// TIA Portal V17 export
// export: Created 2025-05-22T06:00:03.08653Z, ExportSetting WithDefaults, DisplayName Totally Integrated Automation Portal, DisplayVersion V17 Update 8, DisplayName TIA Portal Openness, DisplayVersion V17 Update 8, DisplayName TIA Portal Version Control Interface, DisplayVersion V17, DisplayName SINAMICS Startdrive Advanced, DisplayVersion V17 SP2, DisplayName SINAMICS Startdrive G110M, G120, G120C, G120D, G120P, G115D, DisplayVersion V17 SP2, DisplayName SINAMICS Startdrive G130, G150, S120, S150, SINAMICS MV, S210, DisplayVersion V17 SP2, DisplayName STEP 7 Professional, DisplayVersion V17 Update 8, DisplayName SINUMERIK ONE STEP 7 Toolbox, DisplayVersion V17 Update 12, DisplayName SINUMERIK ONE PLC Basic Program Plus, DisplayVersion V17 Update 12, DisplayName SINUMERIK 840D sl STEP 7 Toolbox, DisplayVersion V17 Update 12, DisplayName STEP 7 Safety, DisplayVersion V17 Update 6, DisplayName WinCC Advanced, DisplayVersion V17 Update 8
FUNCTION "FC421_HOLA_PC_ALARM" : Void   // FC421, LAD
{ S7_Optimized_Access := 'FALSE' }
AUTHOR : ETXETAR
VERSION : 1.0
// stored: AutoNumber false, IsIECCheckEnabled false, SetENOAutomatically false, UDAEnableTagReadback false
   VAR_TEMP
      ERROR : Bool;   // ERROR
      ERROR_CODE : Int;   // ERROR CODE
      ZERO : DWord;   // ZERO
      RESET : Struct   // RESET
         DBB_120 : Word;   // RESET $A_DBB[120]
         DBB_122 : Word;   // RESET $A_DBB[122]
         DBB_124 : Word;   // RESET $A_DBB[124]
         DBB_126 : Word;   // RESET $A_DBB[126]
      END_STRUCT;
   END_VAR
   VAR CONSTANT
      READ : Byte := 16#3;
      WRITE : Byte := 16#4;
      FC_NUMBER : DInt := 202;   // FC NUMBER
   END_VAR
   VAR_TEMP   // added for the SCL form of the ladder/FBD networks
      _w1 : Bool;
      _w2 : Bool;
      _w3 : Bool;
   END_VAR
BEGIN

REGION Network 1: CALL FC21 TOOL ALARMS - $A_DBW[120] TO $A_DBW[126] / READ $A_DBB[102-108]
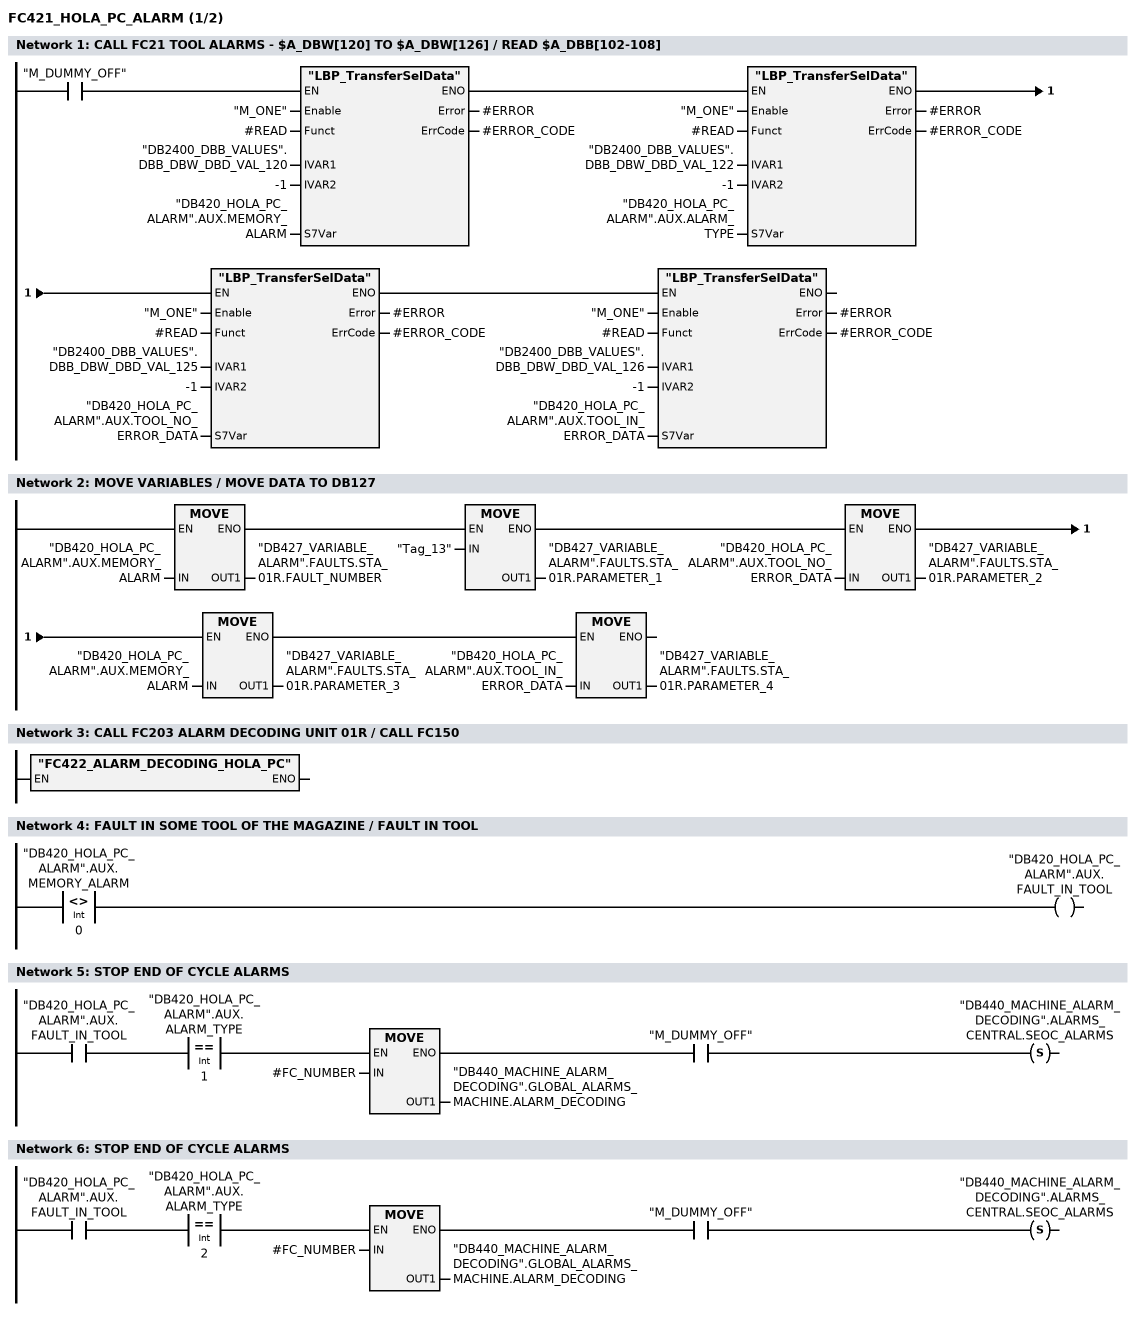
   RUNG wire#powerrail
      Contact( "M_DUMMY_OFF" )
      "LBP_TransferSelData"(Enable := "M_ONE", Funct := #READ, IVAR1 := "DB2400_DBB_VALUES".DBB_DBW_DBD_VAL_120, IVAR2 := -1, S7Var := "DB420_HOLA_PC_ALARM".AUX.MEMORY_ALARM, Error => #ERROR, ErrCode => #ERROR_CODE)
      "LBP_TransferSelData"(Enable := "M_ONE", Funct := #READ, IVAR1 := "DB2400_DBB_VALUES".DBB_DBW_DBD_VAL_122, IVAR2 := -1, S7Var := "DB420_HOLA_PC_ALARM".AUX.ALARM_TYPE, Error => #ERROR, ErrCode => #ERROR_CODE)
      "LBP_TransferSelData"(Enable := "M_ONE", Funct := #READ, IVAR1 := "DB2400_DBB_VALUES".DBB_DBW_DBD_VAL_125, IVAR2 := -1, S7Var := "DB420_HOLA_PC_ALARM".AUX.TOOL_NO_ERROR_DATA, Error => #ERROR, ErrCode => #ERROR_CODE)
      "LBP_TransferSelData"(Enable := "M_ONE", Funct := #READ, IVAR1 := "DB2400_DBB_VALUES".DBB_DBW_DBD_VAL_126, IVAR2 := -1, S7Var := "DB420_HOLA_PC_ALARM".AUX.TOOL_IN_ERROR_DATA, Error => #ERROR, ErrCode => #ERROR_CODE)
   END_RUNG
   // the same network as SCL:
   "LBP_TransferSelData"(EN := "M_DUMMY_OFF",
                         Enable := "M_ONE",
                         Funct := #READ,
                         IVAR1 := "DB2400_DBB_VALUES".DBB_DBW_DBD_VAL_120,
                         IVAR2 := -1,
                         S7Var := "DB420_HOLA_PC_ALARM".AUX.MEMORY_ALARM,
                         Error => #ERROR,
                         ErrCode => #ERROR_CODE,
                         ENO => #_w1);
   "LBP_TransferSelData"(EN := #_w1,
                         Enable := "M_ONE",
                         Funct := #READ,
                         IVAR1 := "DB2400_DBB_VALUES".DBB_DBW_DBD_VAL_122,
                         IVAR2 := -1,
                         S7Var := "DB420_HOLA_PC_ALARM".AUX.ALARM_TYPE,
                         Error => #ERROR,
                         ErrCode => #ERROR_CODE,
                         ENO => #_w2);
   "LBP_TransferSelData"(EN := #_w2,
                         Enable := "M_ONE",
                         Funct := #READ,
                         IVAR1 := "DB2400_DBB_VALUES".DBB_DBW_DBD_VAL_125,
                         IVAR2 := -1,
                         S7Var := "DB420_HOLA_PC_ALARM".AUX.TOOL_NO_ERROR_DATA,
                         Error => #ERROR,
                         ErrCode => #ERROR_CODE,
                         ENO => #_w3);
   IF #_w3 THEN
       "LBP_TransferSelData"(Enable := "M_ONE",
                             Funct := #READ,
                             IVAR1 := "DB2400_DBB_VALUES".DBB_DBW_DBD_VAL_126,
                             IVAR2 := -1,
                             S7Var := "DB420_HOLA_PC_ALARM".AUX.TOOL_IN_ERROR_DATA,
                             Error => #ERROR,
                             ErrCode => #ERROR_CODE);
   END_IF;
END_REGION

REGION Network 2: MOVE VARIABLES / MOVE DATA TO DB127
   RUNG wire#powerrail
      { S7_GenerateENO := "TRUE" } Move(in := "DB420_HOLA_PC_ALARM".AUX.MEMORY_ALARM, out1 => "DB427_VARIABLE_ALARM".FAULTS.STA_01R.FAULT_NUMBER)
      { S7_GenerateENO := "TRUE" } Move(in := "Tag_13", out1 => "DB427_VARIABLE_ALARM".FAULTS.STA_01R.PARAMETER_1)
      { S7_GenerateENO := "TRUE" } Move(in := "DB420_HOLA_PC_ALARM".AUX.TOOL_NO_ERROR_DATA, out1 => "DB427_VARIABLE_ALARM".FAULTS.STA_01R.PARAMETER_2)
      { S7_GenerateENO := "TRUE" } Move(in := "DB420_HOLA_PC_ALARM".AUX.MEMORY_ALARM, out1 => "DB427_VARIABLE_ALARM".FAULTS.STA_01R.PARAMETER_3)
      { S7_GenerateENO := "TRUE" } Move(in := "DB420_HOLA_PC_ALARM".AUX.TOOL_IN_ERROR_DATA, out1 => "DB427_VARIABLE_ALARM".FAULTS.STA_01R.PARAMETER_4)
   END_RUNG
   // the same network as SCL:
   // ENO of a box is taken as its EN; it also drops when the box reports an error
   "DB427_VARIABLE_ALARM".FAULTS.STA_01R.FAULT_NUMBER := "DB420_HOLA_PC_ALARM".AUX.MEMORY_ALARM;
   "DB427_VARIABLE_ALARM".FAULTS.STA_01R.PARAMETER_1 := "Tag_13";
   "DB427_VARIABLE_ALARM".FAULTS.STA_01R.PARAMETER_2 := "DB420_HOLA_PC_ALARM".AUX.TOOL_NO_ERROR_DATA;
   "DB427_VARIABLE_ALARM".FAULTS.STA_01R.PARAMETER_3 := "DB420_HOLA_PC_ALARM".AUX.MEMORY_ALARM;
   "DB427_VARIABLE_ALARM".FAULTS.STA_01R.PARAMETER_4 := "DB420_HOLA_PC_ALARM".AUX.TOOL_IN_ERROR_DATA;
END_REGION

REGION Network 3: CALL FC203 ALARM DECODING UNIT 01R / CALL FC150
   RUNG wire#powerrail
      "FC422_ALARM_DECODING_HOLA_PC"()
   END_RUNG
   // the same network as SCL:
   "FC422_ALARM_DECODING_HOLA_PC"();
END_REGION

REGION Network 4: FAULT IN SOME TOOL OF THE MAGAZINE / FAULT IN TOOL
   RUNG wire#powerrail
      { S7_Templates := "SrcType := Int" } NE_Contact(in1 := "DB420_HOLA_PC_ALARM".AUX.MEMORY_ALARM, in2 := 0)
      Coil( "DB420_HOLA_PC_ALARM".AUX.FAULT_IN_TOOL )
   END_RUNG
   // the same network as SCL:
   "DB420_HOLA_PC_ALARM".AUX.FAULT_IN_TOOL := "DB420_HOLA_PC_ALARM".AUX.MEMORY_ALARM <> 0;
END_REGION

REGION Network 5: STOP END OF CYCLE ALARMS
   RUNG wire#powerrail
      Contact( "DB420_HOLA_PC_ALARM".AUX.FAULT_IN_TOOL )
      { S7_Templates := "SrcType := Int" } EQ_Contact(in1 := "DB420_HOLA_PC_ALARM".AUX.ALARM_TYPE, in2 := 1)
      { S7_GenerateENO := "TRUE" } Move(in := #FC_NUMBER, out1 => "DB440_MACHINE_ALARM_DECODING".GLOBAL_ALARMS_MACHINE.ALARM_DECODING)
      Contact( "M_DUMMY_OFF" )
      S_Coil( "DB440_MACHINE_ALARM_DECODING".ALARMS_CENTRAL.SEOC_ALARMS )
   END_RUNG
   // the same network as SCL:
   // ENO of a box is taken as its EN; it also drops when the box reports an error
   #_w1 := "DB420_HOLA_PC_ALARM".AUX.FAULT_IN_TOOL AND ("DB420_HOLA_PC_ALARM".AUX.ALARM_TYPE = 1);
   IF #_w1 THEN "DB440_MACHINE_ALARM_DECODING".GLOBAL_ALARMS_MACHINE.ALARM_DECODING := #FC_NUMBER; END_IF;
   IF #_w1 AND "M_DUMMY_OFF" THEN "DB440_MACHINE_ALARM_DECODING".ALARMS_CENTRAL.SEOC_ALARMS := TRUE; END_IF;
END_REGION

REGION Network 6: STOP END OF CYCLE ALARMS
   RUNG wire#powerrail
      Contact( "DB420_HOLA_PC_ALARM".AUX.FAULT_IN_TOOL )
      { S7_Templates := "SrcType := Int" } EQ_Contact(in1 := "DB420_HOLA_PC_ALARM".AUX.ALARM_TYPE, in2 := 2)
      { S7_GenerateENO := "TRUE" } Move(in := #FC_NUMBER, out1 => "DB440_MACHINE_ALARM_DECODING".GLOBAL_ALARMS_MACHINE.ALARM_DECODING)
      Contact( "M_DUMMY_OFF" )
      S_Coil( "DB440_MACHINE_ALARM_DECODING".ALARMS_CENTRAL.SEOC_ALARMS )
   END_RUNG
   // the same network as SCL:
   // ENO of a box is taken as its EN; it also drops when the box reports an error
   #_w1 := "DB420_HOLA_PC_ALARM".AUX.FAULT_IN_TOOL AND ("DB420_HOLA_PC_ALARM".AUX.ALARM_TYPE = 2);
   IF #_w1 THEN "DB440_MACHINE_ALARM_DECODING".GLOBAL_ALARMS_MACHINE.ALARM_DECODING := #FC_NUMBER; END_IF;
   IF #_w1 AND "M_DUMMY_OFF" THEN "DB440_MACHINE_ALARM_DECODING".ALARMS_CENTRAL.SEOC_ALARMS := TRUE; END_IF;
END_REGION

REGION Network 7: RESET FAULTS / RESET
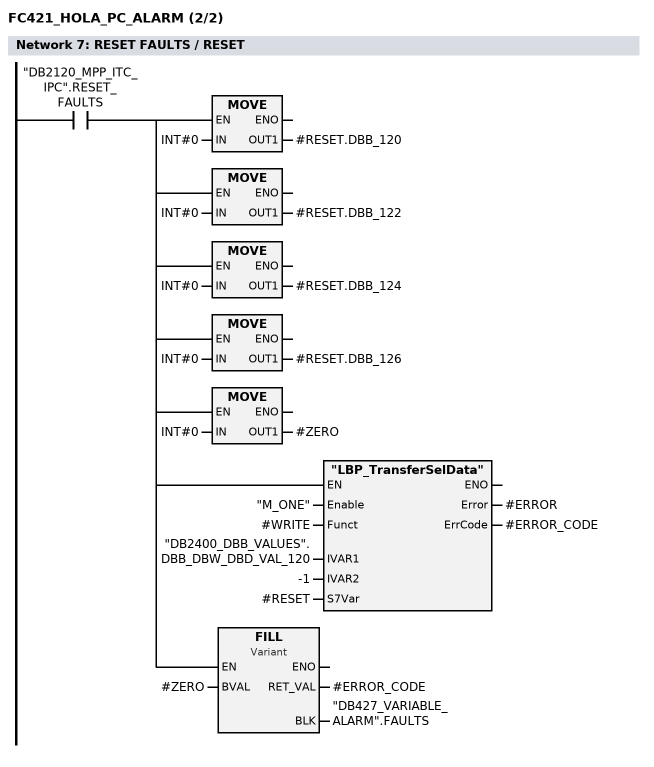
   RUNG wire#powerrail
      Contact( "DB2120_MPP_ITC_IPC".RESET_FAULTS )
      wire#w1
      { S7_GenerateENO := "TRUE" } Move(in := INT#0, out1 => #RESET.DBB_120)
   END_RUNG
   RUNG wire#w1
      { S7_GenerateENO := "TRUE" } Move(in := INT#0, out1 => #RESET.DBB_122)
   END_RUNG
   RUNG wire#w1
      { S7_GenerateENO := "TRUE" } Move(in := INT#0, out1 => #RESET.DBB_124)
   END_RUNG
   RUNG wire#w1
      { S7_GenerateENO := "TRUE" } Move(in := INT#0, out1 => #RESET.DBB_126)
   END_RUNG
   RUNG wire#w1
      { S7_GenerateENO := "TRUE" } Move(in := INT#0, out1 => #ZERO)
   END_RUNG
   RUNG wire#w1
      "LBP_TransferSelData"(Enable := "M_ONE", Funct := #WRITE, IVAR1 := "DB2400_DBB_VALUES".DBB_DBW_DBD_VAL_120, IVAR2 := -1, S7Var := #RESET, Error => #ERROR, ErrCode => #ERROR_CODE)
   END_RUNG
   RUNG wire#w1
      { S7_Templates := "ptr_type := Variant" } FILL(BVAL := #ZERO, RET_VAL => #ERROR_CODE, BLK => "DB427_VARIABLE_ALARM".FAULTS)
   END_RUNG
   // the same network as SCL:
   IF "DB2120_MPP_ITC_IPC".RESET_FAULTS THEN
       #RESET.DBB_120 := INT#0;
       #RESET.DBB_122 := INT#0;
       #RESET.DBB_124 := INT#0;
       #RESET.DBB_126 := INT#0;
       #ZERO := INT#0;
   END_IF;
   #_w1 := "DB2120_MPP_ITC_IPC".RESET_FAULTS;
   IF #_w1 THEN
       "LBP_TransferSelData"(Enable := "M_ONE",
                             Funct := #WRITE,
                             IVAR1 := "DB2400_DBB_VALUES".DBB_DBW_DBD_VAL_120,
                             IVAR2 := -1,
                             S7Var := #RESET,
                             Error => #ERROR,
                             ErrCode => #ERROR_CODE);
       #ERROR_CODE := FILL(BVAL := #ZERO, BLK => "DB427_VARIABLE_ALARM".FAULTS);
   END_IF;
END_REGION
END_FUNCTION
